// Run at the start of each cycle

PROGRAM Fast_Faults_Setup
VAR
END_VAR

g_FastFaultOutput1();

END_PROGRAM

(* stored: Version 1.1.0.1, ProductVersion 3.1.4024.0
   POU Fast_Faults_Setup: Id {bdc9fda1-3ab8-0d1a-09bd-274a15fdc835}, SpecialFunc None *)
